{attribute 'qualified_only'}
{attribute 'strict'}
TYPE ENUM_TestStates :
(
    Unknown := 0,
    OUT := 1,
    TARGET1 := 2,
    TARGET2 := 3
);
END_TYPE

(* stored: Version 1.1.0.1, ProductVersion 3.1.4022.18
   DUT ENUM_TestStates: Id {c258efcc-6b1f-486b-bdf8-0d1ba128e372} *)
